(* IEC 61131-3 sources: GitHub_Test/YF_DoubleAGV/CVC_TcpTest/PLC/DoubleAGV, 7 files *)

(* ---- ClientCalControl_FB.ST ---- *)
FUNCTION_BLOCK ClientCalControl_FB
VAR_EXTERNAL
NDC8 : NDC8_T;
END_VAR

VAR_INPUT

END_VAR

VAR_OUTPUT

END_VAR

VAR
DevDist,IdevDist,Icount,PreDevDist: dint;
P_Scale,I_Scale,D_Scale : real;
PP,PI,PD : real;
P_Curve_Scale,I_Curve_Scale,D_Curve_Scale : real;
PP_Curve,PI_Curve,PD_Curve : real;
FlagCount,OverCount : dint;
Flag : bool;
DevX,PreDevX,DdevDist,ClientX : dint;
PreMasterPositionX,PreMasterPositionY,PreClientPositionX,PreClientPositionY : dint;
AngleScale : real;
END_VAR

if NDC8.OMPLC.GroupFlag=1 and MasterFlag=1 then

	if NDC8.SegmentTrigger.LeftTurn or NDC8.SegmentTrigger.RightTurn then
		FlagCount := 1;

	(*	if dint_to_real(MasterAngle2)/100.0>=(180.0-VV1) and dint_to_real(MasterAngle2)/100.0<=(180.0+VV1) then
			AngleScale := (9496.0/5752.0 - 1.0)/VV1 * abs(abs((dint_to_real(MasterAngle2)/100.0-180.0))-VV1);
		elsif dint_to_real(MasterAngle2)/100.0>=(270.0-VV1) and dint_to_real(MasterAngle2)/100.0<=(270.0+VV1) then
			AngleScale := (9496.0/5752.0 - 1.0)/VV1 * abs(abs((dint_to_real(MasterAngle2)/100.0-270.0))-VV1);
		else
			AngleScale := 0.0;
		end_if;

		if NDC8.SegmentTrigger.Value=1 then
			SegmentAngle := 0;
			if dint_to_real(MasterAngle2)/100.0>=(360.0-VV1) and dint_to_real(MasterAngle2)/100.0<=(0.0+VV1) then
				AngleScale := (9496.0/5752.0 - 1.0)/VV1 * abs(abs((dint_to_real(MasterAngle2)/100.0-180.0))-VV1);
			elsif dint_to_real(MasterAngle2)/100.0>=(90.0-VV1) and dint_to_real(MasterAngle2)/100.0<=(90.0+VV1) then
				AngleScale := (9496.0/5752.0 - 1.0)/VV1 * abs(abs((dint_to_real(MasterAngle2)/100.0-270.0))-VV1);
			else
				AngleScale := 0.0;
			end_if;
		elsif NDC8.SegmentTrigger.Value=2 then
			SegmentAngle := 90;
		elsif NDC8.SegmentTrigger.Value=3 then
			SegmentAngle := 180;
		elsif NDC8.SegmentTrigger.Value=4 then
			SegmentAngle := 270;
		end_if;

		if dint_to_real(MasterAngle2)/100.0>=(180.0-VV1) and dint_to_real(MasterAngle2)/100.0<=(180.0+VV1) then
			AngleScale := (9496.0/5752.0 - 1.0)/VV1 * abs(abs((dint_to_real(MasterAngle2)/100.0-180.0))-VV1);
		elsif dint_to_real(MasterAngle2)/100.0>=(270.0-VV1) and dint_to_real(MasterAngle2)/100.0<=(270.0+VV1) then
			AngleScale := (9496.0/5752.0 - 1.0)/VV1 * abs(abs((dint_to_real(MasterAngle2)/100.0-270.0))-VV1);
		else
			AngleScale := 0.0;
		end_if;*)

		CalculateSpeed := real_to_dint(dint_to_real(MasterSetSpeed)*9496.0/5752.0/(1.0+AngleScale));

		ClientX := real_to_dint(sin(dint_to_real(MasterAngle2)/100.0*3.14159/180.0)*2367.0) + MasterPositionX;

		if MasterAngle2>=9000 and MasterAngle2<=27000 and NDC8.VehicleControl.TravelDir=1 then
			DevX := NDC8.Position.X - ClientX;
		elsif MasterAngle2>=9000 and MasterAngle2<=27000 and NDC8.VehicleControl.TravelDir=0 then
			DevX := ClientX - NDC8.Position.X;
		elsif (MasterAngle2<9000 or MasterAngle2>27000) and NDC8.VehicleControl.TravelDir=1 then
			DevX := ClientX - NDC8.Position.X;
		elsif (MasterAngle2<9000 or MasterAngle2>27000) and NDC8.VehicleControl.TravelDir=0 then
			DevX := NDC8.Position.X - ClientX;
		end_if;

(* --------------------------------PID Adjustment------------------------------------------------- *)
		(* P Adjust *)
		P_Curve_Scale := 0.65;
		PP_Curve := P_Curve_Scale * dint_to_real(DevX);
		if PP_Curve<-150.0 then
			PP_Curve := -150.0;
		elsif PP_Curve>150.0 then
			PP_Curve := 150.0;
		end_if;
		(* I Adjust *)
		if (abs(DevX) > 30)  or Icount > 10 then
			IdevDist := 0;
			Icount := 0;
		else
			IdevDist := DevX + IdevDist;
			Icount := Icount + 1;
		end_if;
		I_Curve_Scale := 0.1;
  		PI_Curve := I_Curve_Scale*dint_to_real(IdevDist);
		if PI_Curve<-20.0 then
			PI_Curve := -20.0;
		elsif PI_Curve>20.0 then
			PI_Curve := 20.0;
		end_if;

		(* D Adjust *)
		if abs(DevX) < 20 then
			DdevDist := DdevDist + DevX - PreDevX ;
		else
			DdevDist := 0;
		end_if;
		PreDevX := DevX;
		PD_Curve := D_Curve_Scale*dint_to_real(DdevDist);
(* --------------------------------PID Adjustment------------------------------------------------- *)

		CalculateSpeed := CalculateSpeed + real_to_dint(PP_Curve+PI_Curve+PD_Curve) ;
		CalculateSpeed := MIN(NDC8.Vehicle.MaxSpeed,CalculateSpeed);

	else

(*	if NDC8.SegmentTrigger.GateOpen then
		if MasterPositionY=PreMasterPositionY then
			;
		else
	 		DevDist := NDC8.Position.Y - MasterPositionY + 4367;
			PreMasterPositionY := MasterPositionY;
		end_if;
	else
		if MasterPositionX=PreMasterPositionX then
			;
		else
	 		DevDist := NDC8.Position.X - MasterPositionX;
			PreMasterPositionX := MasterPositionX;
		end_if;
	end_if;*)

		if NDC8.SegmentTrigger.DirectionY then	(* 两车Y轴方向行驶 *)
			FlagCount := 2;
			if MasterPositionY=PreMasterPositionY then
				;
			else
				if (NDC8.Position.Y-PreClientPositionY)<=0 and (MasterPositionY-PreMasterPositionY)<0 then
			 		DevDist := NDC8.Position.Y - MasterPositionY;
				elsif (NDC8.Position.Y-PreClientPositionY)>=0 and (MasterPositionY-PreMasterPositionY)>0 then
					DevDist := MasterPositionY - NDC8.Position.Y;
				end_if;

				if not Flag then
					Flag := true;
				else
					if abs(DevDist-PreDevDist) > 10 then
						if OverCount > 0 then
							;
						else
					  		DevDist := PreDevDist;
					   	    OverCount := OverCount + 1;
						end_if;
					else
						OverCount := 0;
					end_if;
				end_if;
				PreMasterPositionY := MasterPositionY;
				PreClientPositionY := NDC8.Position.Y;
			end_if;
		else (* 两车X轴方向行驶 *)
			FlagCount := 3;
			if MasterPositionX=PreMasterPositionX then
				;
			else
				if (NDC8.Position.X-PreClientPositionX)<=0 and (MasterPositionX-PreMasterPositionX)<0 then
			 		DevDist := NDC8.Position.X - MasterPositionX;
				elsif (NDC8.Position.X-PreClientPositionX)>=0 and (MasterPositionX-PreMasterPositionX)>0 then
					DevDist := MasterPositionX - NDC8.Position.X;
				end_if;

				if not Flag then
					Flag := true;
				else
					if abs(DevDist-PreDevDist) > 10 then
						if OverCount > 0 then
							;
						else
						   DevDist := PreDevDist;
						   OverCount := OverCount + 1;
						end_if;
					else
						OverCount := 0;
					end_if;
				end_if;

				PreMasterPositionX := MasterPositionX;
				PreClientPositionX := NDC8.Position.X;
			end_if;
	end_if;
	PreDevDist := DevDist;

(* --------------------------------PID Adjustment------------------------------------------------- *)
	(* P Adjust *)
	P_Scale := 0.55;
	PP := P_Scale*dint_to_real(DevDist);
	if PP<-150.0 then
		PP := -150.0;
	elsif PP>150.0 then
		PP := 150.0;
	end_if;
	(* I Adjust *)
	if abs(DevDist) > 10 or Icount > 10 then
		IdevDist := 0;
		Icount := 0;
	else
		IdevDist := DevDist + IdevDist;
		Icount := Icount + 1;
	end_if;
	I_Scale := 0.1;
	PI := I_Scale*dint_to_real(IdevDist);
	if PI<-10.0 then
		PI := -10.0;
	elsif PI>10.0 then
		PI := 10.0;
	end_if;
(* --------------------------------PID Adjustment------------------------------------------------- *)

	CompenstateSpeed := real_to_dint(PP + PI) ;
	end_if;
else
	Flag := false;
	Icount := 0;
	OverCount := 0;
	PreDevDist := 0;
	DevDist := 0;
	DevX := 0;
	CompenstateSpeed := 0;
	CalculateSpeed := 0;
end_if;

END_FUNCTION_BLOCK

(* ---- ClientModeSelect_FB.ST ---- *)
FUNCTION_BLOCK ClientModeSelect_FB
VAR_EXTERNAL
NDC8 : NDC8_T;
END_VAR

VAR_INPUT

END_VAR

VAR_OUTPUT

END_VAR

VAR
ClientVehicleControl : ClientVehicleControl_FB;
ClientCalControl : ClientCalControl_FB;
VirMode,CalMode : bool;
END_VAR

(* 两车组合信号起效且车辆ID等于系统写入的副车ID时，该车变为副车，响应主车的控制 *)
if NDC8.Vehicle.VehicleID=int_to_dint(NDC8.OMPLC.Data10) and MasterFlag=1 and NDC8.OMPLC.GroupFlag=1 then

	if VirMode then	(* 虚拟合体方式 *)
		ClientVehicleControl();
	elsif CalMode then	(* 独立路线跟随方式 *)
		ClientCalControl();
		NDC8.VehicleControl.SlowDown := true;
		if NDC8.SegmentTrigger.LeftTurn or NDC8.SegmentTrigger.RightTurn then
			if CalculateSpeed<80 then
				NDC8.VehicleControl.SlowDownSpeed:= 80;
			else
				NDC8.VehicleControl.SlowDownSpeed:= CalculateSpeed;
			end_if;
		else
			NDC8.VehicleControl.SlowDownSpeed:= MasterSetSpeed + CompenstateSpeed;
		end_if;
	end_if;
end_if;
END_FUNCTION_BLOCK

(* ---- ClientVehicleControl_FB.ST ---- *)
FUNCTION_BLOCK ClientVehicleControl_FB
VAR_EXTERNAL
NDC8 : NDC8_T;
END_VAR

VAR_INPUT

END_VAR

VAR_OUTPUT

END_VAR

VAR

END_VAR

(* 两车组合信号起效且车辆ID等于系统写入的副车ID时，该车变为副车，响应主车的控制 *)
if NDC8.Vehicle.VehicleID=int_to_dint(NDC8.OMPLC.Data10) and MasterFlag=1 and NDC8.OMPLC.GroupFlag=1 then
	(* 使能驱动轮 *)
	NDC8.VehicleControl.PlcSelect := 1;
	NDC8.VehicleControl.PlcSelectMask := 15;
	NDC8.VehicleControl.PlcSetSteerEnable := 1;
	NDC8.VehicleControl.PlcSetDriveEnable := 1;
	(* 关闭LS2000导航 *)
	NDC8.LS2000.NavActive := 0;

	if not HeartBeatTimeOut then (* 确保主副车通讯正常 *)
		NDC8.FrontWheel.PlcSetSpeed := MasterVirFrontSetSpeed;	(* 副车的两轮子速度/角度等于主车的虚拟两轮速度/角度 *)
		NDC8.FrontWheel.PlcSetAngle := MasterVirFrontSetAngle;
		NDC8.RearWheel.PlcSetSpeed  := MasterVirRearSetSpeed;
		NDC8.RearWheel.PlcSetAngle  := MasterVirRearSetAngle;
	else
		NDC8.FrontWheel.PlcSetSpeed := 0;
		NDC8.RearWheel.PlcSetSpeed  := 0;
	end_if;

else
	NDC8.VehicleControl.PlcSelect := 0;
	NDC8.VehicleControl.PlcSelectMask := 0;
	NDC8.VehicleControl.PlcSetSteerEnable := 0;
	NDC8.VehicleControl.PlcSetDriveEnable := 0;

	NDC8.LS2000.NavActive := 1;

	NDC8.UserDefined.VirFrontEncSpeed := NDC8.UserDefined.VirFrontSetSpeed - NDC8.UserDefined.VirFFeedbackSpeed;
	NDC8.UserDefined.VirFrontEncAngle := NDC8.UserDefined.VirFrontSetAngle - NDC8.UserDefined.VirFFeedbackAngle;
	NDC8.UserDefined.VirRearEncSpeed  := NDC8.UserDefined.VirRearSetSpeed - NDC8.UserDefined.VirRFeedbackSpeed;
	NDC8.UserDefined.VirRearEncAngle  := NDC8.UserDefined.VirRearSetAngle - NDC8.UserDefined.VirRFeedbackAngle;
end_if;
END_FUNCTION_BLOCK

(* ---- TcpPort_CRC_FB.ST ---- *)
FUNCTION_BLOCK TcpPort_CRC_FB
VAR_EXTERNAL

END_VAR

VAR_INPUT
cBuffer : ARRAY[1..100] of byte;
CrcLength : uint;
END_VAR

VAR_OUTPUT
CrcHigh: Byte;
CrcLow: Byte;
END_VAR

VAR
i,j : uint ;
wCrc : word ;
wPolynom : word ;
END_VAR
(**************************************************)
wCrc := 16#ffff;
wPolynom := 16#A001;

For I:=3 to CrcLength by 1 do
	wCrc := wCrc xor byte_to_word(cBuffer[I]);
	For J:=0 to 7 by 1 do

		if word_to_bool(wCrc and 16#0001) then
		(*if ROL(wCrc ,15) then*)
			wCrc := SHR(wCrc,1) xor wPolynom;
		else
			wCrc := SHR(wCrc,1);
		end_if;

	end_for;
end_for;
CrcLow := word_to_byte(wCrc);
CrcHigh := word_to_byte( SHR(wCrc,8)  );

END_FUNCTION_BLOCK

(* ---- TcpPortReceive_FB.ST ---- *)
FUNCTION_BLOCK TcpPortReceive_FB
VAR_EXTERNAL
NDC8 : NDC8_T;
END_VAR

VAR_INPUT

END_VAR

VAR_OUTPUT

END_VAR

VAR
serial_read  : NDC8_SERIAL_READ;
TcpPort_CRC : TcpPort_CRC_FB;
PreMasterHeartBeat : dint;
NoHeartBeat : bool;
NoHeartBeatTon : ton;
Count1,index,Count2,TempIndex2,Count3,TempIndex3 : dint;
FirstLength,SecondLength,ThridLength : int;
END_VAR

serial_read(Port:='COM5');
if serial_read.Length>0 then
	Count1 := Count1 + 1;
	FirstLength := serial_read.Length;
	for index:=1 to 32 by 1 do
		TcpPortReceiveDataBytesAll[index] := serial_read.data[index];
	end_for;
end_if;

serial_read(Port:='COM5');
if serial_read.Length>0 then
	Count2 := Count2 + 1;
	SecondLength := serial_read.Length;
	for index:=1 to 32 by 1 do
		TempIndex2 := index + 32;
		TcpPortReceiveDataBytesAll[TempIndex2] := serial_read.data[index];
	end_for;
end_if;

TcpPort_CRC(cBuffer:=TcpPortReceiveDataBytesAll,CrcLength:=53);

if TcpPortReceiveDataBytesAll[1]=16#4A and TcpPortReceiveDataBytesAll[2]=16#54
	and TcpPortReceiveDataBytesAll[54]=TcpPort_CRC.CrcLow and TcpPortReceiveDataBytesAll[55]=TcpPort_CRC.CrcHigh then

	MasterVehicleID := byte_to_dint(TcpPortReceiveDataBytesAll[3]);
	MasterTravelDir := byte_to_dint(TcpPortReceiveDataBytesAll[4]);

	MasterFrontSetSpeed	:= int_to_dint(byte_to_int(TcpPortReceiveDataBytesAll[5])*256 + byte_to_int(TcpPortReceiveDataBytesAll[6]) );

	MasterFrontEncSpeed	:= int_to_dint(byte_to_int(TcpPortReceiveDataBytesAll[7])*256 + byte_to_int(TcpPortReceiveDataBytesAll[8]) );

	MasterFrontSetAngle	:= int_to_dint( byte_to_int(TcpPortReceiveDataBytesAll[9])*256 + byte_to_int(TcpPortReceiveDataBytesAll[10]) );
	MasterFrontEncAngle	:= int_to_dint(byte_to_int(TcpPortReceiveDataBytesAll[11])*256 + byte_to_int(TcpPortReceiveDataBytesAll[12]) );

	MasterRearSetSpeed	:= int_to_dint(byte_to_int(TcpPortReceiveDataBytesAll[13])*256 + byte_to_int(TcpPortReceiveDataBytesAll[14]) );
	MasterRearEncSpeed	:= int_to_dint(byte_to_int(TcpPortReceiveDataBytesAll[15])*256 + byte_to_int(TcpPortReceiveDataBytesAll[16]) );

	MasterRearSetAngle	:= int_to_dint(byte_to_int(TcpPortReceiveDataBytesAll[17])*256 + byte_to_int(TcpPortReceiveDataBytesAll[18]) );
	MasterRearEncAngle	:= int_to_dint(byte_to_int(TcpPortReceiveDataBytesAll[19])*256 + byte_to_int(TcpPortReceiveDataBytesAll[20]) );

	MasterVirFrontSetSpeed	:= int_to_dint(byte_to_int(TcpPortReceiveDataBytesAll[21])*256 + byte_to_int(TcpPortReceiveDataBytesAll[22]) );
	MasterVirFrontEncSpeed	:= int_to_dint(byte_to_int(TcpPortReceiveDataBytesAll[23])*256 + byte_to_int(TcpPortReceiveDataBytesAll[24]) );

	MasterVirFrontSetAngle	:= int_to_dint(byte_to_int(TcpPortReceiveDataBytesAll[25])*256 + byte_to_int(TcpPortReceiveDataBytesAll[26]) );
	MasterVirFrontEncAngle	:= int_to_dint(byte_to_int(TcpPortReceiveDataBytesAll[27])*256 + byte_to_int(TcpPortReceiveDataBytesAll[28]) );

	MasterVirRearSetSpeed	:= int_to_dint(byte_to_int(TcpPortReceiveDataBytesAll[29])*256 + byte_to_int(TcpPortReceiveDataBytesAll[30]) );
	MasterVirRearEncSpeed	:= int_to_dint(byte_to_int(TcpPortReceiveDataBytesAll[31])*256 + byte_to_int(TcpPortReceiveDataBytesAll[32]) );

	MasterVirRearSetAngle	:= int_to_dint(byte_to_int(TcpPortReceiveDataBytesAll[33])*256 + byte_to_int(TcpPortReceiveDataBytesAll[34]) );
	MasterVirRearEncAngle	:= int_to_dint(byte_to_int(TcpPortReceiveDataBytesAll[35])*256 + byte_to_int(TcpPortReceiveDataBytesAll[36]) );

	MasterPositionX := byte_to_dint(TcpPortReceiveDataBytesAll[37])*167777216 + byte_to_dint(TcpPortReceiveDataBytesAll[38])*65536
						+ byte_to_dint(TcpPortReceiveDataBytesAll[39])*256 + byte_to_dint(TcpPortReceiveDataBytesAll[40]) ;

	MasterPositionY := byte_to_dint(TcpPortReceiveDataBytesAll[41])*167777216 + byte_to_dint(TcpPortReceiveDataBytesAll[42])*65536
						+ byte_to_dint(TcpPortReceiveDataBytesAll[43])*256 + byte_to_dint(TcpPortReceiveDataBytesAll[44]) ;

	MasterAngle2 := byte_to_dint(TcpPortReceiveDataBytesAll[45])*256 + byte_to_dint(TcpPortReceiveDataBytesAll[46]) ;

	MasterOpCode  := byte_to_dint(TcpPortReceiveDataBytesAll[47]);
	MasterOpWorking  := byte_to_bool(TcpPortReceiveDataBytesAll[48]);

	MasterSetSpeed := byte_to_dint(TcpPortReceiveDataBytesAll[49])*256 + byte_to_dint(TcpPortReceiveDataBytesAll[50]) ;

	MasterFlag := byte_to_dint(TcpPortReceiveDataBytesAll[51]);

	MasterHeartBeat := byte_to_dint(TcpPortReceiveDataBytesAll[52]);

	MasterErrorStop := byte_to_bool(TcpPortReceiveDataBytesAll[53]);

end_if;

NoHeartBeat := MasterHeartBeat=PreMasterHeartBeat and MasterFlag=1 and NDC8.OMPLC.GroupFlag=1;
NoHeartBeatTon(IN:=NoHeartBeat,PT:=t#2s);
if NoHeartBeatTon.Q then
	HeartBeatTimeOut := true;
else
	HeartBeatTimeOut := false;
end_if;

PreMasterHeartBeat := MasterHeartBeat;

NDC8.UserDefined.HeartBeatTimeOut := HeartBeatTimeOut;
NDC8.UserDefined.MasterErrorStop := MasterErrorStop;

END_FUNCTION_BLOCK

(* ---- TCPPORTSEND_FB.ST ---- *)
FUNCTION_BLOCK TCPPORTSEND_FB
VAR_EXTERNAL
NDC8 : NDC8_T;
END_VAR

VAR_INPUT

END_VAR

VAR_OUTPUT

END_VAR

VAR
serial_write  : NDC8_SERIAL_WRITE;
TcpPort_CRC : TcpPort_CRC_FB;
tempHigh_X,tempHigh_Y,HeartBeat : dint;
ErrorStop,OperationWorking : bool;
index,index1,index2 : dint;
END_VAR

TcpPortSendDataBytesHead[1] := 16#4A;
TcpPortSendDataBytesHead[2] := 16#54;

TcpPortSendDataBytes1[1] := dint_to_byte(NDC8.Vehicle.VehicleID);

TcpPortSendDataBytes1[2] := dint_to_byte(NDC8.VehicleControl.TravelDir);

TcpPortSendDataBytes1[3] := word_to_byte(SHR(dint_to_word(NDC8.UserDefined.FrontSetSpeed),8));
TcpPortSendDataBytes1[4] := dint_to_byte(NDC8.UserDefined.FrontSetSpeed);

TcpPortSendDataBytes1[5] := word_to_byte(SHR(dint_to_word(NDC8.UserDefined.FrontEncSpeed),8));
TcpPortSendDataBytes1[6] := dint_to_byte(NDC8.UserDefined.FrontEncSpeed);

TcpPortSendDataBytes1[7] := word_to_byte(SHR(dint_to_word(NDC8.UserDefined.FrontSetAngle),8));
TcpPortSendDataBytes1[8] := dint_to_byte(NDC8.UserDefined.FrontSetAngle);

TcpPortSendDataBytes1[9] := word_to_byte(SHR(dint_to_word(NDC8.UserDefined.FrontEncAngle),8));
TcpPortSendDataBytes1[10] := dint_to_byte(NDC8.UserDefined.FrontEncAngle);

TcpPortSendDataBytes1[11] := word_to_byte(SHR(dint_to_word(NDC8.UserDefined.RearSetSpeed),8));
TcpPortSendDataBytes1[12] := dint_to_byte(NDC8.UserDefined.RearSetSpeed);

TcpPortSendDataBytes1[13] := word_to_byte(SHR(dint_to_word(NDC8.UserDefined.RearEncSpeed),8));
TcpPortSendDataBytes1[14] := dint_to_byte(NDC8.UserDefined.RearEncSpeed);

TcpPortSendDataBytes1[15] := word_to_byte(SHR(dint_to_word(NDC8.UserDefined.RearSetAngle),8));
TcpPortSendDataBytes1[16] := dint_to_byte(NDC8.UserDefined.RearSetAngle);

TcpPortSendDataBytes1[17] := word_to_byte(SHR(dint_to_word(NDC8.UserDefined.RearEncAngle),8));
TcpPortSendDataBytes1[18] := dint_to_byte(NDC8.UserDefined.RearEncAngle);

TcpPortSendDataBytes1[19] := word_to_byte(SHR(dint_to_word(NDC8.UserDefined.VirFrontSetSpeed),8));
TcpPortSendDataBytes1[20] := dint_to_byte(NDC8.UserDefined.VirFrontSetSpeed);

TcpPortSendDataBytes1[21] := word_to_byte(SHR(dint_to_word(NDC8.UserDefined.VirFrontEncSpeed),8));
TcpPortSendDataBytes1[22] := dint_to_byte(NDC8.UserDefined.VirFrontEncSpeed);

TcpPortSendDataBytes1[23] := word_to_byte(SHR(dint_to_word(NDC8.UserDefined.VirFrontSetAngle),8));
TcpPortSendDataBytes1[24] := dint_to_byte(NDC8.UserDefined.VirFrontSetAngle);

TcpPortSendDataBytes1[25] := word_to_byte(SHR(dint_to_word(NDC8.UserDefined.VirFrontEncAngle),8));
TcpPortSendDataBytes1[26] := dint_to_byte(NDC8.UserDefined.VirFrontEncAngle);

TcpPortSendDataBytes1[27] := word_to_byte(SHR(dint_to_word(NDC8.UserDefined.VirRearSetSpeed),8));
TcpPortSendDataBytes1[28] := dint_to_byte(NDC8.UserDefined.VirRearSetSpeed);

TcpPortSendDataBytes1[29] := word_to_byte(SHR(dint_to_word(NDC8.UserDefined.VirRearEncSpeed),8));
TcpPortSendDataBytes1[30] := dint_to_byte(NDC8.UserDefined.VirRearEncSpeed);

TcpPortSendDataBytes1[31] := word_to_byte(SHR(dint_to_word(NDC8.UserDefined.VirRearSetAngle),8));
TcpPortSendDataBytes1[32] := dint_to_byte(NDC8.UserDefined.VirRearSetAngle);

TcpPortSendDataBytes2[1] := word_to_byte(SHR(dint_to_word(NDC8.UserDefined.VirRearEncAngle),8));
TcpPortSendDataBytes2[2] := dint_to_byte(NDC8.UserDefined.VirRearEncAngle);

tempHigh_X := NDC8.Position.X / 65536;
TcpPortSendDataBytes2[3] := word_to_byte(SHR(dint_to_word(tempHigh_X),8));
TcpPortSendDataBytes2[4] := dint_to_byte(tempHigh_X);
TcpPortSendDataBytes2[5] := word_to_byte(SHR(dint_to_word(NDC8.Position.X),8));
TcpPortSendDataBytes2[6] := dint_to_byte(NDC8.Position.X);

tempHigh_Y := NDC8.Position.Y / 65536;
TcpPortSendDataBytes2[7] := word_to_byte(SHR(dint_to_word(tempHigh_Y),8));
TcpPortSendDataBytes2[8] := dint_to_byte(tempHigh_Y);
TcpPortSendDataBytes2[9] := word_to_byte(SHR(dint_to_word(NDC8.Position.Y),8));
TcpPortSendDataBytes2[10] := dint_to_byte(NDC8.Position.Y);

TcpPortSendDataBytes2[11] := word_to_byte(SHR(dint_to_word(NDC8.Position.Angle2),8));
TcpPortSendDataBytes2[12] := dint_to_byte(NDC8.Position.Angle2);

TcpPortSendDataBytes2[13] := dint_to_byte(NDC8.LoadOperation.OperationCode);
TcpPortSendDataBytes2[14] := bool_to_byte(OperationWorking);

TcpPortSendDataBytes2[15] := word_to_byte(SHR(dint_to_word(NDC8.VehicleControl.SetSpeed),8));
TcpPortSendDataBytes2[16] := dint_to_byte(NDC8.VehicleControl.SetSpeed);

TcpPortSendDataBytes2[17] := int_to_byte(NDC8.OMPLC.GroupFlag);

TcpPortSendDataBytes2[18] := dint_to_byte(HeartBeat);

TcpPortSendDataBytes2[19] := bool_to_byte(ErrorStop);

For index:=1 to 2 by 1 do
	TcpPortSendDataBytesAll[index] := TcpPortSendDataBytesHead[index];
end_for;

For index:=3 to 34 by 1 do
	index1 := index - 2 ;
	TcpPortSendDataBytesAll[index] := TcpPortSendDataBytes1[index1];
end_for;

For index:=35 to 53 by 1 do
	index2 := index - 34 ;
	TcpPortSendDataBytesAll[index] := TcpPortSendDataBytes2[index2];
end_for;

TcpPort_CRC(cBuffer:=TcpPortSendDataBytesAll,CrcLength:=53);
TcpPortSendDataBytesCrc[1] := TcpPort_CRC.CrcLow;
TcpPortSendDataBytesCrc[2] := TcpPort_CRC.CrcHigh;

serial_write( port:='COM5',data:=TcpPortSendDataBytesHead,length:=2 );
serial_write( port:='COM5',data:=TcpPortSendDataBytes1,length:=32 );
serial_write( port:='COM5',data:=TcpPortSendDataBytes2,length:=19 );
serial_write( port:='COM5',data:=TcpPortSendDataBytesCrc,length:=2 );
serial_write( port:='COM5',data:=TcpPortSendDataBytesHead,length:=0 );

if HeartBeat=0 then
	HeartBeat := 1;
elsif HeartBeat=1 then
	HeartBeat := 0;
end_if;

ErrorStop := NDC8.VehicleControl.Stop or NDC8.VehicleControl.EStop or NDC8.VehicleControl.QuickStop
				or NDC8.CanOpenMaster.NMTState<>5 or NDC8.CanOpenMaster.State<>0 ;

(*OperationWorking := OUTPUT.PlatRaise and NDC8.VehicleControl.OperationMode=0;*)

END_FUNCTION_BLOCK

(* ---- UPDATEFEEDBACK_FB.ST ---- *)
FUNCTION_BLOCK UPDATEFEEDBACK_FB
VAR_EXTERNAL
NDC8 : NDC8_T;
END_VAR

VAR_INPUT

END_VAR

VAR_OUTPUT

END_VAR

VAR
TimerBlink : blink;
END_VAR

TimerBlink(CYCLE :=t#100ms,RUN:=true);

NDC8.UserDefined.VirFFeedbackSpeed := bool_to_dint(TimerBlink.Q1) + 1;
NDC8.UserDefined.VirRFeedbackSpeed := bool_to_dint(TimerBlink.Q1) + 1;
NDC8.UserDefined.VirFFeedbackAngle := bool_to_dint(TimerBlink.Q1) + 1;
NDC8.UserDefined.VirRFeedbackAngle := bool_to_dint(TimerBlink.Q1) + 1;

END_FUNCTION_BLOCK
